# EPICS alarm handler configuration: mps_database/bareTest/alarms/areas/mpln_ltus_mp04.alhConfig
GROUP NULL MPLN:LTUS:MP04:1
$ALIAS MPS Link Node 206
$GUIDANCE
LTUH MPS
   Group Name: MPLN:LTUS:MP04:1
   Summary PV:  MPLN:LTUS:MP04:1:STATSUMY
$END
CHANNEL  MPLN:LTUS:MP04:1    MPLN:LTUS:MP04:1:MPS_EN_RBV		-----
CHANNEL  MPLN:LTUS:MP04:1    MPLN:LTUS:MP04:1:LC1_MODE_RBV		-----
